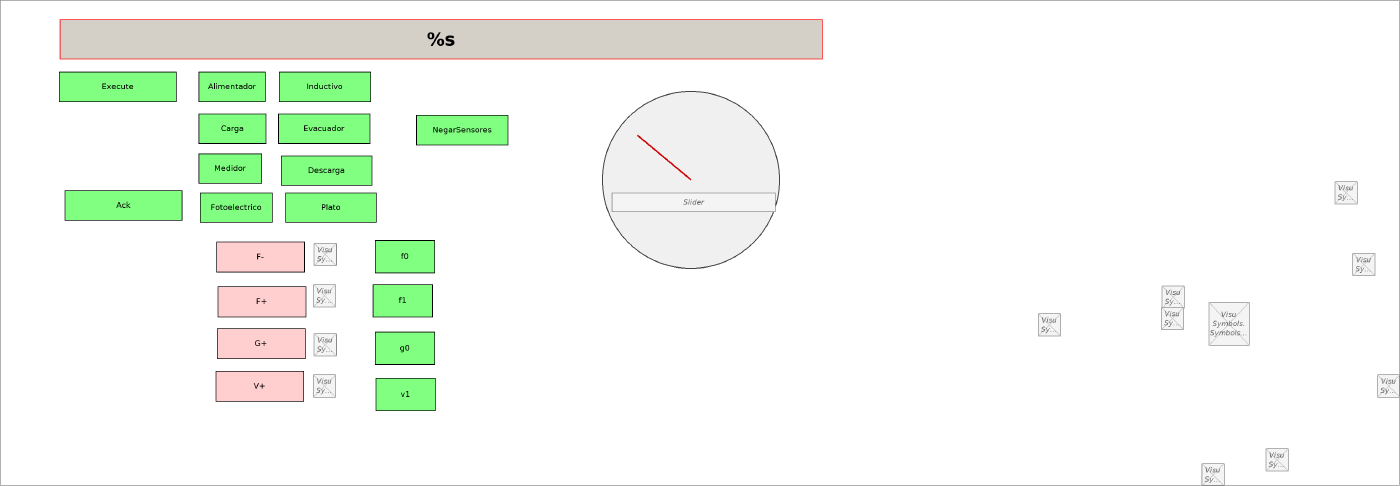
VISUALIZATION FMS205Testing  // 1968x684
VAR_IN_OUT
	
END_VAR
(*VAR
	TestAlimentador
END_VAR^*)
    Meter180 (846,128 250x250), value: MAIN.fbFMS205.fbPanel.cn.NewSpeed, style: Meter-Meter180-Gray, scale format: %.1f, scale 0..200
    Rectangle (84,27 1072x56), "%s", text variable: sel(MAIN.fbFMS205.fbPanel.Probando,'Panel de pruebas inactivo','Panel de pruebas ACTIVO')
        toggle MAIN.fbFMS205.fbPanel.Probando
    Rectangle (83,101 165x42), "Execute"
        toggle MAIN.fbFMS205.td.Execute
    Rectangle (91,268 165x42), "Ack"
        tap MAIN.fbFMS205.td.Ack
    Rectangle (279,101 94x42), "Alimentador"
        toggle MAIN.fbFMS205.td.Alime
    Rectangle (279,160 95x42), "Carga"
        toggle MAIN.fbFMS205.td.Carga
    Rectangle (279,216 89x42), "Medidor"
        toggle MAIN.fbFMS205.td.Medid
    Rectangle (281,271 102x42), "Fotoelectrico"
        toggle MAIN.fbFMS205.td.Fotoe
    Rectangle (392,101 129x42), "Inductivo"
        toggle MAIN.fbFMS205.td.Induc
    Rectangle (391,160 129x42), "Evacuador"
        toggle MAIN.fbFMS205.td.Evacu
    Rectangle (395,219 128x42), "Descarga"
        toggle MAIN.fbFMS205.td.Desca
    Rectangle (401,271 128x42), "Plato"
        toggle MAIN.fbFMS205.td.Plato
    Rectangle (585,162 129x42), "NegarSensores"
        tap MAIN.fbFMS205.td.Negar
    Slider (860,271 230x27), variable: MAIN.fbFMS205.fbPanel.cn.NewSpeed, scale 1..200
    Image (1699,425 57x61), image: VisuSymbols.Symbols.ArrowHalfLeftUp
    Image (1876,255 32x32), image: VisuSymbols.Symbols.ArrowQuarterRightLeft
    Image (1901,356 32x32), image: VisuSymbols.Symbols.ArrowBoldUp
    Image (441,469 32x32), invisible if: MAIN.fbFMS205.mdEvacuador.G_1.uiInvisible, image: VisuSymbols.Symbols.ArrowBoldDown
        p2773130477: MAIN.fbFMS205.mdEvacuador.G_1.UIDown
    Image (1633,402 32x32), image: VisuSymbols.Symbols.BatteryFull
    Image (1632,432 32x32), image: VisuSymbols.Symbols.Lock
    Image (440,527 32x32), invisible if: MAIN.fbFMS205.mdEvacuador.V_1.uiInvisible, image: VisuSymbols.Symbols.4ArrowsIn
        p2858320360: MAIN.fbFMS205.mdEvacuador.V_1.uiClockwise
    Image (441,342 32x32), invisible if: MAIN.fbFMS205.mdEvacuador.F_0.uiInvisible, image: VisuSymbols.Symbols.ArrowBoldLeft
        p3528305787: MAIN.fbFMS205.mdEvacuador.F_0.uiLeft
    Image (440,400 32x32), invisible if: MAIN.fbFMS205.mdEvacuador.F_1.uiInvisible, image: VisuSymbols.Symbols.ArrowBoldRight
        p3528305787: MAIN.fbFMS205.mdEvacuador.F_1.uiRight
    Image (1936,527 32x32), image: VisuSymbols.Symbols.ArrowBoldRightUp
    Image (1689,652 32x32), image: VisuSymbols.Symbols.ArrowQuarterRightDown
    Image (1779,631 32x32), image: VisuSymbols.Symbols.ArrowQuarterLeftUp
    Image (1459,441 32x32), image: VisuSymbols.Symbols.ArrowBoldRightDown
    Rectangle (305,462 124x43), "G+", tooltip "tooltip generada", input disabled if: MAIN.fbFMS205.mdEvacuador.G_1.uiEnabled
        toggle MAIN.fbFMS205.mdEvacuador.G_1.uiValue
    Rectangle (303,522 124x43), "V+", tooltip "tooltip generada", input disabled if: MAIN.fbFMS205.mdEvacuador.V_1.uiEnabled
        toggle MAIN.fbFMS205.mdEvacuador.V_1.uiValue
    Rectangle (306,403 124x43), "F+", tooltip "tooltip generada", input disabled if: MAIN.fbFMS205.mdEvacuador.F_1.uiEnabled
        toggle MAIN.fbFMS205.mdEvacuador.F_1.uiValue
    Rectangle (524,400 84x46), "f1"
        toggle MAIN.fbFMS205.mdEvacuador.f1.uiValue
    Rectangle (304,340 124x43), "F-", tooltip "tooltip generada", input disabled if: MAIN.fbFMS205.mdEvacuador.F_0.uiEnabled
        toggle MAIN.fbFMS205.mdEvacuador.F_0.uiValue
    Rectangle (527,338 84x46), "f0"
        toggle MAIN.fbFMS205.mdEvacuador.f0.uiValue
    Rectangle (527,467 84x46), "g0"
        toggle MAIN.fbFMS205.mdEvacuador.g0.uiValue
    Rectangle (528,532 84x46), "v1"
        toggle MAIN.fbFMS205.mdEvacuador.v1.uiValue
END_VISUALIZATION

(* stored: Version 1.1.0.1, ProductVersion 3.1.4024.11
   Visu FMS205Testing: Id {d10fef3f-e567-4db8-8634-f52f25296e47} *)
